Yaskawa INFORM job: R1_W02,4,6(0_0)_KM-OK.JBI

/JOB
//NAME R1_W02,4,6(0_0)_KM-OK
///FOLDERNAME SCIANA-NOWY-R2-KM
//POS
///NPOS 77,77,0,4,0,0
///TOOL 0
///POSTYPE PULSE
///PULSE
C00000=-174522,6583,732,-81114,57384,-11781
C00001=-172960,12703,8525,-82305,58217,-10791
C00002=-173420,13658,9390,-82287,57878,-10798
C00003=-172960,12703,8525,-82305,58217,-10791
C00004=-172483,14222,9903,-82389,58551,-10725
C00005=-172960,12703,8525,-82305,58217,-10791
C00006=-174088,5167,5264,-84729,55731,-9256
C00007=-171280,11849,6984,-89376,52288,-7705
C00008=-171280,12128,8246,-89869,52259,-7340
C00009=-171280,11849,6984,-89376,52288,-7705
C00010=-176368,5115,10483,-94107,48535,-4388
C00011=-161133,-21431,-11620,-32290,31717,38951
C00012=-166193,-13735,-2683,-28322,28551,36737
C00013=-166365,-11916,-1340,-28035,28588,36586
C00014=-166193,-13735,-2683,-28322,28551,36737
C00015=-166484,-12796,-826,-28573,27869,36854
C00016=-166193,-13735,-2683,-28322,28551,36737
C00017=-161927,-24594,-12798,-32484,31998,39256
C00018=-155155,-6207,-30499,-23040,84085,41474
C00019=-187974,16007,-465,-74860,68606,-73739
C00020=-187971,16014,-459,-74861,68608,-73738
C00021=-187970,16017,-457,-74861,68609,-73738
C00022=-188065,16322,-175,-74847,68538,-73741
C00023=-187970,16017,-457,-74861,68609,-73738
C00024=-187982,15993,-478,-74858,68601,-73740
C00025=-188123,15688,-759,-74825,68507,-73762
C00026=-187982,15993,-478,-74858,68601,-73740
C00027=-187982,15995,-476,-74858,68601,-73740
C00028=-188055,16230,-74,-74890,68512,-73687
C00029=-187982,15995,-476,-74858,68601,-73740
C00030=-187983,15992,-479,-74858,68601,-73740
C00031=-185123,16527,-5629,-74315,71577,-75055
C00032=-165643,5472,-22008,-57816,82906,-32840
C00033=-153600,-19645,-23752,-41320,66430,4214
C00034=-161010,6792,897,-39431,61770,2600
C00035=-161008,6803,906,-39432,61771,2600
C00036=-161074,6865,1159,-39463,61645,2620
C00037=-161075,4879,-316,-39487,61556,2657
C00038=-160508,6816,-113,-39396,62494,2543
C00039=-160959,7092,1492,-34589,61222,1662
C00040=-157931,14438,8425,-38644,65989,5471
C00041=-155353,20308,15528,-39705,66096,6633
C00042=-153350,7555,1346,-39668,68707,6522
C00043=-174436,-11399,3906,-23747,38202,33405
C00044=-174416,-11363,3933,-23761,38209,33414
C00045=-155155,-6207,-30499,-23040,84085,41474
C00046=-167856,42942,44479,-44576,87949,75494
C00047=-174201,39824,30698,-44830,89717,71735
C00048=-174202,39772,30629,-44830,89729,71730
C00049=-174300,38678,29865,-44827,89618,71734
C00050=-173753,38726,28593,-44851,90472,71609
C00051=-173790,41778,32604,-44829,89804,71890
C00052=-174440,38939,30130,-43450,86434,69208
C00053=-174625,39116,29841,-43438,86538,69076
C00054=-174452,38184,29186,-43444,86567,69141
C00055=-174215,39612,30410,-43455,86673,69209
C00056=-163437,11239,19048,-64558,76519,55979
C00057=-172819,4226,12636,-64344,70595,54342
C00058=-171600,10063,21711,-65155,70219,55665
C00059=-171586,11063,23159,-65273,70065,55836
C00060=-170302,17238,32521,-66069,69775,57175
C00061=-167466,13624,23757,-64976,73158,56067
C00062=-174214,39663,30476,-43455,86662,69214
C00063=-166320,47562,38864,-43573,89751,71531
C00064=-155155,-6207,-30499,-23040,84085,41474
C00065=-158532,-24414,-4804,-32267,22916,49173
C00066=-162219,-15798,1425,-26285,22163,46063
C00067=-160659,-10505,5478,-28325,22871,47138
C00068=-160667,-11361,4484,-25333,18870,47058
C00069=-161098,-12444,3311,-27327,23025,46629
C00070=-159658,-10599,5699,-29947,23053,47982
C00071=-160762,-11077,5021,-25395,18673,47081
C00072=-160738,-11186,5373,-25787,18434,47269
C00073=-160661,-10807,5180,-25528,18740,47150
C00074=-160656,-10808,5155,-25519,18754,47146
C00075=-135615,-20366,-13260,-37178,48093,50762
C00076=-15978,-102434,-83816,-28834,48298,44128
BC00000=389371,883224,717072
BC00001=378707,895443,708103
BC00002=378707,895443,708103
BC00003=378707,895443,708103
BC00004=378707,895443,708103
BC00005=378707,895443,708103
BC00006=378034,890325,685589
BC00007=375161,868470,589450
BC00008=375161,868470,589447
BC00009=375161,868470,589450
BC00010=390381,882138,667249
BC00011=303246,823192,856112
BC00012=303246,823192,856112
BC00013=303246,823192,856112
BC00014=303246,823192,856112
BC00015=303246,823192,856112
BC00016=303246,823192,856112
BC00017=303924,826322,868010
BC00018=297455,809016,882806
BC00019=389426,843654,667560
BC00020=384481,838451,656958
BC00021=382502,836370,652718
BC00022=380113,836348,652712
BC00023=382502,836370,652718
BC00024=391231,834561,627737
BC00025=391255,832257,627761
BC00026=391231,834561,627737
BC00027=389247,835739,621366
BC00028=389248,835732,613301
BC00029=389247,835739,621366
BC00030=391225,837820,625606
BC00031=396171,843023,636208
BC00032=360773,830829,724635
BC00033=314255,821989,864432
BC00034=314255,821989,864432
BC00035=308132,825470,852305
BC00036=305756,826822,847596
BC00037=305683,826863,847454
BC00038=305683,826863,847454
BC00039=309405,830338,834596
BC00040=309405,830338,834596
BC00041=309405,830338,834596
BC00042=309405,830338,834596
BC00043=333968,867875,937281
BC00044=333921,867878,1044815
BC00045=297455,809016,882806
BC00046=334185,798105,989913
BC00047=334134,798292,882381
BC00048=331405,792594,866884
BC00049=330314,790315,860686
BC00050=330314,790315,860686
BC00051=330314,790315,860686
BC00052=334605,784967,862717
BC00053=352171,785134,809076
BC00054=352171,785134,809076
BC00055=353454,787302,815346
BC00056=356663,792718,831017
BC00057=356663,792718,831017
BC00058=356663,792718,831017
BC00059=356663,792718,831017
BC00060=356663,792718,831017
BC00061=356663,792718,831017
BC00062=356663,792720,831020
BC00063=356713,792534,938552
BC00064=297455,809016,882806
BC00065=302565,831732,1074843
BC00066=302515,831918,967310
BC00067=295799,835067,957970
BC00068=290675,829418,930260
BC00069=293112,836327,954234
BC00070=293112,836327,954234
BC00071=290675,829418,930260
BC00072=290745,817286,842643
BC00073=293384,815876,846102
BC00074=299979,812352,854751
BC00075=300030,812166,962284
BC00076=278008,791254,977380
///POSTYPE BASE
///RECTAN
///RCONF 0,0,0,0,0,0,0,0,0,0,0,0,0,0,0,0,0,0,0,0,0,0,0,0
P00006=0.222,-3.123,-1.508,0.0000,0.0000,0.0000
P00021=-0.225,-6.128,-0.405,0.0000,0.0000,0.0000
P00024=0.145,-0.552,1.326,0.0000,0.0000,0.0000
P00026=0.562,-0.002,-0.337,0.0000,0.0000,0.0000
//INST
///DATE 2024/07/17 17:57
///ATTR SC,RW
///GROUP1 RB1,BS1
NOP
SFTOF
MOVL C00000 BC00000 V=333.3
MOVL C00001 BC00001 V=166.7
REFP 3 C00002 BC00002
CALL JOB:SEARCH-R1
SET P021 P006
SFTON P021
MOVL C00003 BC00003 V=60.0
REFP 3 C00004 BC00004
CALL JOB:SEARCH-R1
SET P021 P006
SFTON P021
MOVL C00005 BC00005 V=166.7
MOVL C00006 BC00006 V=166.7
MOVL C00007 BC00007 V=166.7
REFP 3 C00008 BC00008
CALL JOB:SEARCH-R1
SET P021 P006
SFTON P021
MOVL C00009 BC00009 V=166.7
MOVL C00010 BC00010 V=100.0
SFTOF
MOVL C00011 BC00011 V=166.7
MOVL C00012 BC00012 V=166.7
REFP 3 C00013 BC00013
CALL JOB:SEARCH-R1
SET P026 P006
SFTON P026
MOVL C00014 BC00014 V=60.0
REFP 3 C00015 BC00015
CALL JOB:SEARCH-R1
SET P026 P006
SFTON P026
MOVL C00016 BC00016 V=60.0
MOVL C00017 BC00017 V=250.0
MOVJ C00018 BC00018 VJ=100.00
'Path S705 (for W3)
SFTOF
MOVL C00019 BC00019 V=166.7
MOVL C00020 BC00020 V=250.0
MOVL C00021 BC00021 V=250.0
REFP 3 C00022 BC00022
CALL JOB:SEARCH-R1
SET P024 P006
SFTON P024
MOVL C00023 BC00023 V=166.7
MOVL C00024 BC00024 V=166.7
REFP 3 C00025 BC00025
CALL JOB:SEARCH-R1
SET P024 P006
SFTON P024
MOVL C00026 BC00026 V=166.7
MOVL C00027 BC00027 V=166.7
REFP 3 C00028 BC00028
CALL JOB:SEARCH-R1
SET P024 P006
SFTON P024
MOVL C00029 BC00029 V=166.7
MOVL C00030 BC00030 V=166.7
MOVL C00031 BC00031 V=166.7
MOVJ C00032 BC00032 VJ=100.00
MOVJ C00033 BC00033 VJ=100.00
'Path W1
SFTOF
SFTON P026
MOVL C00034 BC00034 V=166.7
MOVL C00035 BC00035 V=166.7
MOVL C00036 BC00036 V=166.7 PL=0
REFP 1 C00037 BC00037
REFP 2 C00038 BC00038
MACRO1 MJ#(0) ARGF10
ARCON
MOVL C00039 BC00039 V=13.3
MOVL C00040 BC00040 V=13.3
MOVL C00041 BC00041 V=13.3
ARCOF
SFTOF
MOVL C00042 BC00042 V=250.0
'Path W2
SFTOF
SFTON P021
MOVL C00043 BC00043 V=250.0
MOVL C00044 BC00044 V=250.0
SFTOF
'
MOVJ C00045 BC00045 VJ=100.00
'Path W786
SFTOF
SFTON P024
MOVJ C00046 BC00046 VJ=100.00
MOVL C00047 BC00047 V=250.0
MOVL C00048 BC00048 V=166.7
MOVL C00049 BC00049 V=166.7 PL=0
REFP 1 C00050 BC00050
REFP 2 C00051 BC00051
MACRO1 MJ#(0) ARGF10
ARCON
MOVL C00052 BC00052 V=13.3
MOVL C00053 BC00053 V=13.3
MOVL C00054 BC00054 V=11.7
ARCOF
MOVL C00055 BC00055 V=166.7
SFTOF
MOVL C00056 BC00056 V=333.3
MACRO1 MJ#(0) ARGF7
MOVL C00057 BC00057 V=250.0
ARCON
MOVL C00058 BC00058 V=11.7
MOVL C00059 BC00059 V=11.7
MOVL C00060 BC00060 V=11.7
ARCOF
MOVL C00061 BC00061 V=166.7
MOVL C00062 BC00062 V=250.0
MOVL C00063 BC00063 V=250.0
SFTOF
MOVJ C00064 BC00064 VJ=100.00
'
'Path W4
SFTOF
SFTON P021
MOVJ C00065 BC00065 VJ=100.00
MOVL C00066 BC00066 V=333.3
MOVL C00067 BC00067 V=250.0
MOVL C00068 BC00068 V=166.7 PL=0
REFP 1 C00069 BC00069
REFP 2 C00070 BC00070
MACRO1 MJ#(0) ARGF10
ARCON
MOVL C00071 BC00071 V=13.3
MOVL C00072 BC00072 V=13.3
ARCOF
MOVL C00073 BC00073 V=166.7
MOVL C00074 BC00074 V=250.0
MOVJ C00075 BC00075 VJ=100.00
MOVJ C00076 BC00076 VJ=100.00
SFTOF
END
